{attribute 'qualified_only'}
VAR_GLOBAL
	AxisHMI_1: ST_HMI_Axis;
	bMoveRel : BOOL;
	bMoveVel : BOOL;
	bStop : BOOL;
END_VAR

(* stored: Version 1.1.0.1, ProductVersion 3.1.4024.0
   GVL gHMI: Id {e027e335-39c7-4ca5-9ca8-66eb092a49c3} *)
